KUKA KRL program: sps.sub

&ACCESS RVP
&REL 1
&COMMENT 03-10-R1 SUBMIT SPS
&PARAM DISKPATH = System
DEF  SPS ( )
   ;FOLD DECLARATIONS
  ;FOLD BASISTECH DECL
  ;Automatic External
  DECL STATE_T STAT
  DECL MODUS_T MODE
  ;ENDFOLD (BASISTECH DECL)
  ;FOLD USER DECL
  ; Please insert user defined declarations

  ;ENDFOLD (USER DECL)
  ;ENDFOLD (DECLARATIONS)
  ;FOLD INI
  ;FOLD AUTOEXT INIT
  INTERRUPT DECL 91 WHEN $PRO_STATE1==#P_FREE DO RESET_OUT ()
  INTERRUPT ON 91
  $LOOP_MSG[]="                                                            "
  MODE=#SYNC
  $H_POS=$H_POS
  ;Automatic External: IN EXTERNAL AUTOMATIC MODE SELECT THE MAIN PROGRAM /R1/CELL()
  IF $MODE_OP==#EX THEN
    CWRITE($CMD,STAT,MODE,"RUN /R1/CELL()")
  ENDIF
  ;ENDFOLD (AUTOEXT INIT)
  ;FOLD BACKUPMANAGER PLC INIT
  BM_ENABLED = FALSE
  BM_OUTPUTVALUE = 0
  ;ENDFOLD (BACKUPMANAGER PLC INIT)
  ;FOLD TQM_INIT
    TorqueDefinitions()
  ;ENDFOLD (TQM_INIT)



  ;FOLD USER INIT
  ; Please insert user defined initialization commands

  ;ENDFOLD (USER INIT)
  ;ENDFOLD (INI)
;********************************
; Gestamp Standards
; Line - BMW G65 (cell 03)
; Robot 03-10-R1 (BMW-03-10-R1)
; Application - SUBMIT INTERPRETER (BACKGROUND LOGIC, CENTERLINE SENSORS, NUT PRELOAD)
;********************************

  LOOP
    WAIT FOR NOT($POWER_FAIL)
    TORQUE_MONITORING()
    ;FOLD BACKUPMANAGER PLC
    IF BM_ENABLED THEN
      BM_OUTPUTSIGNAL = BM_OUTPUTVALUE
    ENDIF
    ;ENDFOLD (BACKUPMANAGER PLC)
;START AUTOGENERATED -- DO NOT CHANGE -- GripperSpotTech sps SpsSub.add InsertGripperTechGlobals
    ;FOLD GRIPPERTECH LOOP
      GRPg_ChkSetStatePLC()
   ;ENDFOLD (GRIPPERTECH LOOP)
;END AUTOGENERATED -- DO NOT CHANGE -- (GripperSpotTech sps SpsSub.add InsertGripperTechGlobals)
;NOTE: THE CALL NutWeld_BKG() WAS COMMENTED OUT IN THE ARCHIVE, THE FOLD BELOW IS EMPTY: NO HOPPER
;NOTE: LEVEL LIGHTS $OUT[477]/$OUT[478],
;NOTE: NO NUTWELD STATUS KEYS AND NO NUTWELD PROCESS RESET ON PROGRAM CANCEL (F12, F29)
;FOLD NutWeld PLC
;ENDFOLD (NutWeld PLC)
;NOTE: THE CALL AutomationCore_BKG() WAS COMMENTED OUT IN THE ARCHIVE, THE FOLD BELOW IS EMPTY -
;NOTE: ITS PLC STATUS BITS STAY STATIC (F12, C01)
;FOLD Automation Core PLC
;ENDFOLD (Automation Core PLC)

			;FOLD Centerline Pedestal
   ;NOTE: INTEGRATOR CODE FOR THE CENTERLINE PEDESTAL NUT WELDER, RUN IN EVERY SUBMIT CYCLE


	;GUN STROKE POSITION (BALLUFF BTL6 LPT) - SIGNALS $IN[567..590] CL_LPT_BYTE1..3 INTO
	;CL_GunStrokePositionLPT, BYTE ORDER HIGH TO LOW: BYTE1, BYTE2, BYTE3 (BYTE0 IS NOT USED);
	;CENTERLINE_WELD CHECKS IT (GUN ON THE NUT 69000..73000, GUN OPEN > 120000)
	;CHECK: R20 BUILDS THE SAME VALUE FROM ALL FOUR BYTES IN ANOTHER ORDER - CONFIRM THE BTL6
	;CHECK: OUTPUT FORMAT ON THIS PEDESTAL (F23)
	CL_GunStrokePositionLPT=(CL_LPT_BYTE1*65536)+(CL_LPT_BYTE2*256)+CL_LPT_BYTE3

   ;UPPER PIN POSITION - SIGNALS $IN[591..606] CL_PIN_BYTE0..1 INTO CL_WeldPinPosition
   ;NOTE: NO PROGRAM READS CL_WeldPinPosition - THE PIN POSITIONS ARE NOT CHECKED (F16)
   CL_WeldPinPosition=(CL_PIN_BYTE0*256)+CL_PIN_BYTE1

   ;WATER FLOW SV0500 - SIGNALS $IN[3000..3015] SV0500_BYTE0..1 INTO SV0500_FLOW
   SV0500_FLOW =( SV0500_BYTE0*256)+SV0500_BYTE1

   ;CL_WaterOk = TRUE WHEN SV0500_FLOW > 1230, ELSE FALSE; NOTHING READS CL_WaterOk
   ;WARNING: dipw1_WaterOk (A BOOL VARIABLE, NOT A SIGNAL) IS SET TRUE IN BOTH BRANCHES - THE
   ;  WATER FLOW RESULT IS THROWN AWAY. CENTERLINE_WELD DOES NOT READ EITHER ONE (F09)
   ;CHECK: OLD COMMENT SAID "1230 = WATER OK", BUT THE CODE TREATS EXACTLY 1230 AS NOT OK (F09)
   IF SV0500_FLOW > 1230 THEN
   CL_WaterOk = TRUE
   dipw1_WaterOk = TRUE
   ELSE
   CL_WaterOk = FALSE
   dipw1_WaterOk = TRUE
   ENDIF

   ;KL50L2 BEACON - SIGNALS $OUT[3008] CL_BeaconBit3008 (BYTE 589 BIT 0),
   ;$OUT[3024] CL_BeaconBit3024 (BYTE 591 BIT 0), $OUT[3001] CL_BeaconBit3001 (NOT MAPPED ON THE BUS)
   ;NOTE: NONE OF THE BITS IS EVER SWITCHED OFF EXCEPT $OUT[3024]. $OUT[478]/$OUT[477] ARE WRITTEN
   ;NOTE: ONLY BY NutWeld_Bkg, WHICH IS DISABLED: THIS BLOCK NEVER SWITCHES THE BEACON (F29)
   ;RED: WHEN SIGNAL $OUT[478] dopw1_LowLevel ON - SIGNALS $OUT[3008] CL_BeaconBit3008 ON,
   ;$OUT[3024] CL_BeaconBit3024 ON
    IF dopw1_LowLevel THEN
     CL_BeaconBit3008 = TRUE
     CL_BeaconBit3024 = TRUE
    ENDIF
   ;GREEN: WHEN SIGNAL $OUT[477] dopw1_LevelOk ON - SIGNALS $OUT[3001] CL_BeaconBit3001 ON,
   ;$OUT[3024] CL_BeaconBit3024 OFF
   ;CHECK: $OUT[3001] IS NOT MAPPED; R20 USES $OUT[3000] AND $OUT[3016] FOR THE SAME BEACON (F29)
    IF  dopw1_LevelOk THEN
     CL_BeaconBit3001 = TRUE
     CL_BeaconBit3024 = FALSE
    ENDIF


;ENDFOLD (Centerline Pedestal)

   ;COOLING WATER ON - SIGNAL $OUT[475] dopw1_StartWater ON WHILE SIGNAL $IN[4] di004UseDryCycle OFF
   ;NOTE: WRITTEN IN EVERY SUBMIT CYCLE AND NEVER SWITCHED OFF HERE: IT OVERRIDES THE WATER OFF
   ;NOTE: OF CENTERLINE_HOME AND DOES NOT USE SIGNAL $IN[13] di013WaterEnable (F09)
IF di004UseDryCycle==FALSE THEN
   dopw1_StartWater=TRUE
   ENDIF

   ;NUT PRELOAD SEQUENCE (Program/Centerline/PRELOAD.src): SWITCHES THE PEDESTAL VALVES
   ;$OUT[471..505] AND SETS NUT_READY; STARTED BY NUT_START (MOTION TRIGGERS IN PICK/WELD APPS)
   ;WARNING: RUNS IN EVERY OPERATING MODE (ALSO T1/T2, NO ENABLING SWITCH) AND WRITES THE SAME
   ;WARNING: VALVES AS THE ROBOT PROGRAMS, WITH NO OWNERSHIP BETWEEN THEM (F11)
PRELOAD()

    ;FOLD USER PLC
    ;Make your modifications here

    ;ENDFOLD (USER PLC)
  ENDLOOP
  ;FOLD ;%{H}
  ;FOLD
END
  ;ENDFOLD


;NOTE: RESET_OUT RUNS WHEN THE ROBOT PROGRAM IS CANCELLED ($PRO_STATE1 = #P_FREE) AND ONLY RESETS
;NOTE: THE PGNO HANDSHAKE OUTPUTS - THE CENTERLINE PEDESTAL IS NOT PUT IN A SAFE STATE (F10)
DEF  RESET_OUT ( )
  INT N
  MsgLoop(" ")
  IF REFLECT_PROG_NR == 1 THEN
    FOR N = 0 TO PGNO_LENGTH - 1
      $OUT[PGNO_FBIT_REFL + N] = FALSE
    ENDFOR
  ENDIF
  IF (PGNO_REQ>0) THEN
    $OUT[PGNO_REQ]=FALSE
  ELSE
    IF (PGNO_REQ<0) THEN
      $OUT[-PGNO_REQ]=TRUE
    ENDIF
  ENDIF
END

;FOLD USER SUBROUTINE
; Integrate your user defined subroutines

;ENDFOLD (USER SUBROUTINE)
;ENDFOLD
